// TIA Portal V17 export
// export: Created 2021-12-03T08:13:09.3443444Z, ExportSetting WithDefaults, DisplayName Totally Integrated Automation Portal, DisplayVersion V17, DisplayName TIA Portal Openness, DisplayVersion V17, DisplayName TIA Portal Version Control Interface, DisplayVersion V17, DisplayName STEP 7 Professional, DisplayVersion V17, DisplayName STEP 7 Safety, DisplayVersion V17, DisplayName WinCC Advanced, DisplayVersion V17
FUNCTION "FFC_Reintegration" : Void   // FC302, F_FBD
AUTHOR : TSe
VERSION : 0.1
// Реинтеграция Failsafe модулей
// stored: AutoNumber false, IsIECCheckEnabled false, UDAEnableTagReadback false
BEGIN

REGION Network 1: Reset
   // Запрос на сброс по нажатию синей кнопки или через HMI
END_REGION

REGION Network 2: Reintegration after Communication/Channel-Error at the F-DO
   // In case of passivation a positive flank on ACK_REI is necessary. For this 
   // acknowledgement the memory bit REINT is prepared.
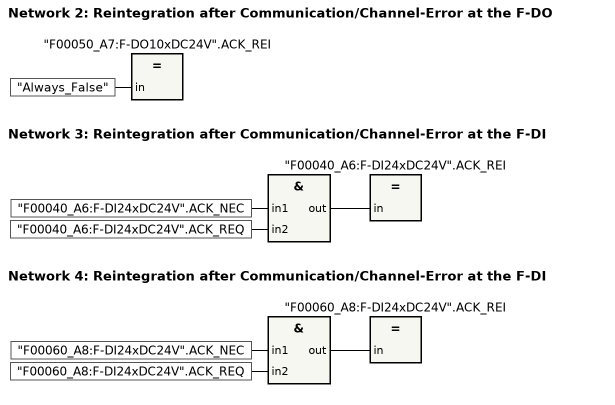
   "F00050_A7:F-DO10xDC24V".ACK_REI := "Always_False";
END_REGION

REGION Network 3: Reintegration after Communication/Channel-Error at the F-DI
   // If ACK_NEC="1" a positive flank on ACK_REI is necessary. This is possible only, 
   // if ACK_REQ="1". ACK_REQ="1" will be set by the system (in the case of a 
   // dissapeared error). After this the system reset ACK_REQ.
   "F00040_A6:F-DI24xDC24V".ACK_REI := "F00040_A6:F-DI24xDC24V".ACK_NEC AND "F00040_A6:F-DI24xDC24V".ACK_REQ;
END_REGION

REGION Network 4: Reintegration after Communication/Channel-Error at the F-DI
   // If ACK_NEC="1" a positive flank on ACK_REI is necessary. This is possible only, 
   // if ACK_REQ="1". ACK_REQ="1" will be set by the system (in the case of a 
   // dissapeared error). After this the system reset ACK_REQ.
   "F00060_A8:F-DI24xDC24V".ACK_REI := "F00060_A8:F-DI24xDC24V".ACK_NEC AND "F00060_A8:F-DI24xDC24V".ACK_REQ;
END_REGION
END_FUNCTION
